TYPE stInput :
STRUCT
	start	:	BOOL;
	stop	:	BOOL;
	emg		:	BOOL;
	ack		:	BOOL;
	FC1		:	BOOL;
	FC2		:	BOOL;	
END_STRUCT
END_TYPE

(* stored: Version 1.1.0.1
   DUT stInput: Id {f1dd25d7-0ea3-02f8-348d-7450be40006b} *)
